PROGRAM AntiBlockingPump
VAR
	fbHVACAntiBlockingPump: FB_HVACAntiBlockingPump;
	eDataSecurityType: E_HVACDataSecurityType := E_HVACDataSecurityType.eHVACDataSecurityType_Idle;
	bSetDefault: BOOL;
	bEnable: BOOL;
	bDisable: BOOL;
	bIn: BOOL;
	dtSystemTime: DATE_AND_TIME;
	bReset: BOOL;
	eAntiBlockingMode: E_HVACAntiBlockingMode;
	iHoursDowntime: INT;
	iDayWeekly: INT;
	iHour: INT;
	iMinute: INT;
	iLenghtImpulse: INT;
	bOut: BOOL;
	bOutAndAntiBlocking: BOOL;
	bQAntiBlocking: BOOL;
	bInvalidParameter: BOOL;
END_VAR

fbHVACAntiBlockingPump(
	eDataSecurityType:=eDataSecurityType, 
	bSetDefault:=bSetDefault, 
	bEnable:=bEnable, 
	bDisable:=bDisable, 
	bIn:=bIn, 
	dtSystemTime:=dtSystemTime, 
	bReset:=bReset, 
	eAntiBlockingMode:=eAntiBlockingMode, 
	iHoursDowntime:=iHoursDowntime, 
	iDayWeekly:=iDayWeekly, 
	iHour:=iHour, 
	iMinute:=iMinute, 
	iLenghtImpulse:=iLenghtImpulse, 
	bOut=>bOut, 
	bOutAndAntiBlocking=>bOutAndAntiBlocking, 
	bQAntiBlocking=>bQAntiBlocking, 
	bInvalidParameter=>bInvalidParameter);

END_PROGRAM

(* stored: Version 1.1.0.1, ProductVersion 3.1.4024.4
   POU AntiBlockingPump: Id {39b28447-0fe7-43dd-ad6f-709d33adec0a}, SpecialFunc None *)
